{attribute 'linkalways'} 
{attribute 'no_explicit_call' := 'This FB is a CLASS and must be accessed using methods or properties'}
{attribute 'enable_dynamic_creation'}
FUNCTION_BLOCK Node_F_VN_DrawContours EXTENDS Node
VAR
    ipContours : _ITcVnContainer;
    nContourIndex : _DINT(0);
    ipDestImage : _ITcVnImage;
    //aColor _TcVnVector4_LREAL;
    nThickness : _DINT(1);
    hrPrev : _HRESULT(S_OK);
	hresult : _HRESULT(S_OK);
END_VAR

METHOD PUBLIC  Clone : I_Node
VAR
	pNode : POINTER TO Node_F_VN_DrawContours
;
END_VAR
pNode := __NEW(Node_F_VN_DrawContours
);
Clone := pNode^;
END_METHOD

METHOD FB_init : BOOL
VAR_INPUT
	bInitRetains : BOOL; // if TRUE, the retain variables are initialized (warm start / cold start)
	bInCopyCode : BOOL;  // if TRUE, the instance afterwards gets moved into the copy code (online change)
END_VAR
AddInput('ipContours', ipContours);
AddInput('nContourIndex', nContourIndex);
AddInput('ipDestImage', ipDestImage);
AddInput('hrPrev', hrPrev);
AddOutput('ipDestImage', ipDestImage);
AddOutput('hresult',hresult);
AddParameter('nThickness', nThickness);
END_METHOD

METHOD PROTECTED  OnExecute : HRESULT

//REMOVE
VAR
    aColor_Green : TcVnVector4_LREAL := [0, 255, 0, 0];
END_VAR
hresult.Value := F_VN_DrawContours(
    ipContours := ipContours.Value,
    nContourIndex := nContourIndex.Value,
	ipDestImage := ipDestImage.Value,
    aColor := aColor_Green,
    nThickness := nThickness.Value,
	hrPrev:= hrPrev.Value);
END_METHOD

END_FUNCTION_BLOCK

(* stored: Version 1.1.0.1, ProductVersion 3.1.4024.13
   POU Node_F_VN_DrawContours: Id {35a4fce0-ca9c-0ac1-30e1-7d017faab450}, SpecialFunc None
   Folder Constructor: Id {e2d56749-f117-057b-2676-31b8b2dfb507}
   Method Clone: Id {3116d9a6-5586-02ad-1613-b2178a2c362f}
   Method FB_init: Id {09d529d7-292e-0e7e-3a63-470dbaff2f70}
   Method OnExecute: Id {ef1597a4-9cfe-058a-226a-4fbb85125199} *)
